{attribute 'strict'}
TYPE COLOR :
(
	AZUL := 2,
	VERDE := 5,
	METAL := 8,
	VACIO := 0
);
END_TYPE

(* stored: Version 1.1.0.1, ProductVersion 3.1.4024.12
   DUT COLOR: Id {67ca2d69-dc13-42d5-bbd6-721edda9390d} *)
